TYPE ACRMemoryUIntEvent EXTENDS ACRMemoryEvent :
STRUCT
	_Value : UINT;
END_STRUCT
END_TYPE

(* stored: Version 1.1.0.1, ProductVersion 3.1.4020.12
   DUT ACRMemoryUIntEvent: Id {697a795c-4be4-448d-9e3f-760cd40cba4a} *)
